// TIA Portal V20 export
DATA_BLOCK "DB_OPC_Maintenance"   // DB93
{ S7_Optimized_Access := 'TRUE' }
// stored: MemoryReserve 100
   VAR
      NumberOfTasks : Int := 16;
      Tasks : Array[0..100] of "UDT_OPC_Maintenance";
   END_VAR
BEGIN
END_DATA_BLOCK
